// TIA Portal V16 export
// export: Created 2022-02-09T12:08:03.87452Z, ExportSetting WithDefaults, DisplayName Totally Integrated Automation Portal, DisplayVersion V16 Update 5, DisplayName TIA Portal Version Control Interface, DisplayVersion V16 Update 2, DisplayName TIA Portal Openness, DisplayVersion V16 Update 5, DisplayName STEP 7 Professional, DisplayVersion V16 Update 5, DisplayName STEP 7 Safety, DisplayVersion V16, DisplayName WinCC Professional, DisplayVersion V16 Update 5, DisplayName SIMATIC Visualization Architect, DisplayVersion V16
DATA_BLOCK "TEST_EV_Aireacio"   // DB2
{ S7_Optimized_Access := 'TRUE' }
VERSION : 0.1
// stored: AutoNumber true, DBAccessibleFromOPCUA true, IsOnlyStoredInLoadMemory false, IsRetainMemResEnabled false, IsWriteProtectedInAS false, MemoryReserve 100
   VAR
      aPosTra_Auto : Bool;
      psEnaAutoGrl : "boto";
      psEnaManualGrl { S7_SetPoint := 'True'} : "boto";
      psResetAlarma { S7_SetPoint := 'True'} : "boto";
   END_VAR
BEGIN
END_DATA_BLOCK
